Fanuc KAREL source: kb00023.KL

-- PROVISIONAL review KL for V940-1; original PC SHA256 07dbd8adbf538d650c01cced00fb4de398f0c32088565b1b19b8822f8ea3f4aa
-- Incomplete behavior may be omitted. Consult companion uncertainty JSON. Do not deploy.
PROGRAM KB00023
%NOLOCKGROUP
BEGIN
  -- V9_ZERO_TABLE_METADATA_HINT layout=0002_ascii; no indexed target words; source/name/runtime held
  -- UNRESOLVED_PC offsets 5-12; opcodes 9D,23
  -- UNRESOLVED_PC offsets 17-24; opcodes 9D,23
  -- UNRESOLVED_PC offsets 29-45; opcodes 27,22,22,31
  -- UNRESOLVED_PC offsets 50-54; opcodes 7F
END KB00023
